{attribute 'linkalways'} 
{attribute 'no_explicit_call' := 'This FB is a CLASS and must be accessed using methods or properties'}
{attribute 'enable_dynamic_creation'}
FUNCTION_BLOCK Node_F_VN_ApproximatePolygon EXTENDS VisionNode
VAR
    ipSrcContour : _ITcVnContainer;
    ipDestContour : _ITcVnContainer;
    fMaxDist : _LREAL(0.0);
    bClosed : _BOOL(FALSE);
    hrPrev : _HRESULT(S_OK);
	hresult : _HRESULT(S_OK);
END_VAR

METHOD PUBLIC  Clone : I_Node
VAR
	pNode : POINTER TO Node_F_VN_ApproximatePolygon;
END_VAR
pNode := __NEW(Node_F_VN_ApproximatePolygon);
Clone := pNode^;
END_METHOD

METHOD FB_init : BOOL
VAR_INPUT
	bInitRetains : BOOL; // if TRUE, the retain variables are initialized (warm start / cold start)
	bInCopyCode : BOOL;  // if TRUE, the instance afterwards gets moved into the copy code (online change)
END_VAR
AddInput('ipSrcContour', ipSrcContour);
AddParameter('fMaxDist', fMaxDist);
AddParameter('bClosed', bClosed);
AddInput('hrPrev', hrPrev);
AddOutput('ipDestContour', ipDestContour);
AddOutput('hresult',hresult);
END_METHOD

METHOD PROTECTED OnExecute
hresult.Value := F_VN_ApproximatePolygon(
	ipSrcContour := ipSrcContour.Value,
    ipDestContour := ipDestContour.Value,
    fMaxDist := fMaxDist.Value,
    bClosed := bClosed.Value,
	hrPrev:= hrPrev.Value);
END_METHOD

METHOD PUBLIC PreExecutionCheck
VAR_INPUT
	Check : I_PreExecutionChecks;
END_VAR
Check.IsTrue(ipSrcContour.IsValid, 'ipSrcContour must be a valid container');
Check.IsTrue((ipSrcContour.IsType(TC_GLOBAL_CONST_LIST.ContainerType_Vector_TcVnPoint2_DINT) OR
              ipSrcContour.IsType(TC_GLOBAL_CONST_LIST.ContainerType_Vector_TcVnPoint2_REAL)),
              'ipSrcContour contains incorrect type');
END_METHOD

END_FUNCTION_BLOCK

(* stored: Version 1.1.0.1, ProductVersion 3.1.4026.13
   POU Node_F_VN_ApproximatePolygon: Id {46d1f5da-16bb-003f-2827-7db044f73b16}, SpecialFunc None
   Folder Constructor: Id {747268f7-ade1-0c9e-0d1d-baeea9b20513}
   Method Clone: Id {3c21cf3d-cb45-0281-21b7-2be34affbc8b}
   Method FB_init: Id {4ab56b67-7a52-0743-1baf-ccfce23c404f}
   Method OnExecute: Id {907fda12-a089-0f16-2437-832bec1abe8b}
   Method PreExecutionCheck: Id {4555ba28-153b-0e48-19b5-32d1e1949046} *)
